% RSLogix 500 project converyor.RSS, saved by version 8.30.00.16 %
PROJECT "UNTITLED"    % processor: Bul.1763 MicroLogix 1100 Series B %

PROGRAM FILES
  LAD 2 "MAIN"  2 rungs
  LAD 3 "I/O"  8 rungs

DATA FILES
  O0 OUTPUT  5 elements
  I1 INPUT  7 elements
  S2 STATUS  66 elements
  B3 BINARY  1 elements
  T4 TIMER  1 elements
  C5 COUNTER  1 elements
  R6 CONTROL  1 elements
  N7 INTEGER  1 elements
  F8 FLOAT  1 elements

LADDER 2 "MAIN"
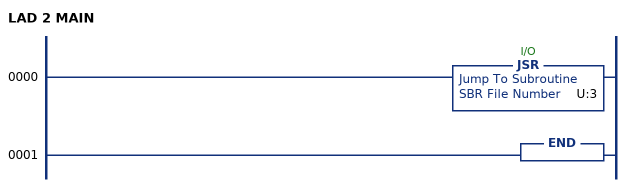
% Rung: 0 %
SOR JSR U:3 EOR
%   U:3  "I/O" %
% Rung: 1 %
SOR END EOR

LADDER 3 "I/O"
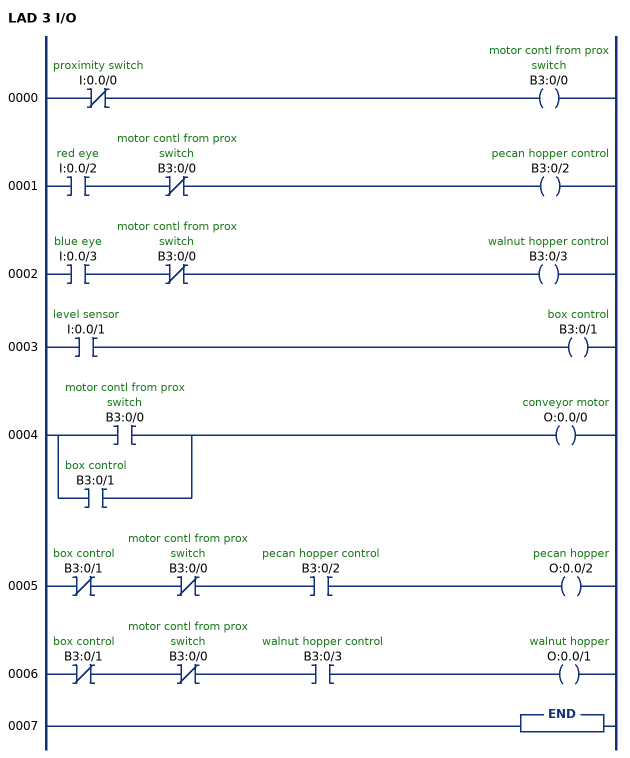
% Rung: 0 %
SOR XIO I:0.0/0 OTE B3:0/0 EOR
%   I:0.0/0  "proximity switch" %
%   B3:0/0  "motor contl from prox switch" %
% Rung: 1 %
SOR XIC I:0.0/2 XIO B3:0/0 OTE B3:0/2 EOR
%   I:0.0/2  "red eye" %
%   B3:0/0  "motor contl from prox switch" %
%   B3:0/2  "pecan hopper control" %
% Rung: 2 %
SOR XIC I:0.0/3 XIO B3:0/0 OTE B3:0/3 EOR
%   I:0.0/3  "blue eye" %
%   B3:0/0  "motor contl from prox switch" %
%   B3:0/3  "walnut hopper control" %
% Rung: 3 %
SOR XIC I:0.0/1 OTE B3:0/1 EOR
%   I:0.0/1  "level sensor" %
%   B3:0/1  "box control" %
% Rung: 4 %
SOR BST XIC B3:0/0 NXB XIC B3:0/1 BND OTE O:0.0/0 EOR
%   B3:0/0  "motor contl from prox switch" %
%   B3:0/1  "box control" %
%   O:0.0/0  "conveyor motor" %
% Rung: 5 %
SOR XIO B3:0/1 XIO B3:0/0 XIC B3:0/2 OTE O:0.0/2 EOR
%   B3:0/1  "box control" %
%   B3:0/0  "motor contl from prox switch" %
%   B3:0/2  "pecan hopper control" %
%   O:0.0/2  "pecan hopper" %
% Rung: 6 %
SOR XIO B3:0/1 XIO B3:0/0 XIC B3:0/3 OTE O:0.0/1 EOR
%   B3:0/1  "box control" %
%   B3:0/0  "motor contl from prox switch" %
%   B3:0/3  "walnut hopper control" %
%   O:0.0/1  "walnut hopper" %
% Rung: 7 %
SOR END EOR

OTHER DOCUMENTED ADDRESSES
  U:4  "controls"
